(* IEC 61131-3 sources: ATCMcontrol_Engineering/src/COM/softing/fc/CL/Libs/ATCM_IEC1131_3/table_24, 7 files *)

(* ---- add.st ---- *)
(*[[
    UserURL= "ATCMFile:ADD.htm"
]]*)

FUNCTION ADD : ANY_MAGNITUDE
VAR_INPUT
    IN1 : ANY_MAGNITUDE;
END_VAR
VAR_IN_EXT
    IN2 : ANY_MAGNITUDE;
END_VAR

inline +

END_FUNCTION

(* ---- div.st ---- *)
(*[[
    UserURL= "ATCMFile:DIV.htm"
]]*)

FUNCTION DIV : ANY_NUM
VAR_INPUT
    IN1: ANY_NUM;
    IN2: ANY_NUM;
END_VAR

inline /

END_FUNCTION

(* ---- expt.st ---- *)
(*[[
    UserURL= "ATCMFile:EXPT.htm"
]]*)

FUNCTION EXPT : ANY_REAL
VAR_INPUT
    IN1: ANY_REAL;
    IN2: ANY_NUM;
END_VAR

inline **

END_FUNCTION

(* ---- mod.st ---- *)
(*[[
    UserURL= "ATCMFile:MOD.htm"
]]*)

FUNCTION MOD : ANY_INT
VAR_INPUT
    IN1: ANY_INT;
    IN2: ANY_INT;
END_VAR

inline MOD

END_FUNCTION

(* ---- move.st ---- *)
(*[[
    UserURL= "ATCMFile:MOVE.htm"
]]*)

FUNCTION MOVE: ANY
VAR_INPUT
    In: ANY;
END_VAR

inline :=

END_FUNCTION

(* ---- mul.st ---- *)
(*[[
    UserURL= "ATCMFile:MUL.htm"
]]*)

FUNCTION MUL : ANY_NUM
VAR_INPUT
    IN1 : ANY_NUM;
END_VAR
VAR_IN_EXT
    IN2 : ANY_NUM;
END_VAR

inline *

END_FUNCTION

(* ---- sub.st ---- *)
(*[[
    UserURL= "ATCMFile:SUB.htm"
]]*)

FUNCTION SUB : ANY_MAGNITUDE
VAR_INPUT
    IN1: ANY_MAGNITUDE;
    IN2: ANY_MAGNITUDE;
END_VAR

inline -

END_FUNCTION
